PROGRAM MAIN
VAR
    axis: AXIS_REF;
    fbAxisPower: MC_Power;
    //fbAxisMoveAbsolute: MC_MoveAbsolute;
    
	bEnable: BOOL := TRUE;
    fOverride: LREAL := 100;
    	
	biLimFwd_AirRoll AT %I*: BOOL;
	biLimBwd_AirRoll AT %I*: BOOL;
	
	biLimFwd_CrysGap AT %I*: BOOL;
	biLimBwd_CrysGap AT %I*: BOOL;
	
END_VAR

axis.ReadStatus();
(*

fbAxisPower(
    Axis:= axis,
    Enable:= bEnable,
    Enable_Positive:= biLimFwd_AirRoll,
    Enable_Negative:= biLimBwd_AirRoll,
    Override:= fOverride,
    BufferMode:= ,
    Options:= ,
    Status=> ,
    Busy=> ,
    Active=> ,
    Error=> ,
    ErrorID=> );
	*)

END_PROGRAM

(* stored: Version 1.1.0.1, ProductVersion 3.1.4024.4
   POU MAIN: Id {3931aef3-4867-4d88-b736-03fecad4f8a1}, SpecialFunc None *)
